FUNCTION_BLOCK FB_Test
VAR_INPUT
END_VAR
VAR_OUTPUT
END_VAR
VAR
	nCallCount : UINT;
	nB : ARRAY[0..2] OF INT;
END_VAR

{attribute 'TcRpcEnable' := '1'}
METHOD M_Test : BOOL
VAR_INPUT
	a : INT;
	b : ARRAY[0..2] OF INT;
END_VAR
nCallCount := nCallCount + 1;
nB[0] := b[0];
nB[1] := b[1];
nB[2] := b[2];
M_Test := TRUE;
END_METHOD

END_FUNCTION_BLOCK

(* stored: Version 1.1.0.1, ProductVersion 3.1.4024.3
   POU FB_Test: Id {f96d368f-e17a-4b3d-b947-64c3790d4dca}, SpecialFunc None
   Method M_Test: Id {4842830d-928e-4d21-97ca-29dd587d9088} *)
